(* Logix 5000 project; controller new_PLC_2 vendor 1 type 14 code 235 rev 37.11; software revision 37.00 *)

TASK MainTask (continuous, watchdog 500 ms) : MainProgram
TASK SafetyTask (periodic, rate 20 ms, priority 10, watchdog 20 ms, safety) : SafetyProgram

MODULES
   Local : vendor 1 type 14 code 235 (5069 0, rev 37.11)
      Tarjeta_Ethernet : vendor 1 type 12 code 200 (Ethernet 10.12.143.10, rev 10.7, Output RPI 10 ms)
           Point_IO_Gabinete_4:4:I   // Sensor Lane Change -
           Point_IO_Gabinete_2:4:O.3   // Stack Light Red
           Point_IO_Gabinete_2:4:O.1   // Stack Light Orange
           Point_IO_Gabinete_2:4:O.2   // Stack Light Green
           Point_IO_Gabinete_2:4:O   // Storage 2 Outputs Stack Lights
           Point_IO_Gabinete_4:8:O.2   // Cognex Light 2
           Point_IO_Gabinete_4:8:O.0   // Main Valve
           Point_IO_Gabinete_4:8:O.3   // Cognex Light 1
           Point_IO_Gabinete_4:8:O   // Main valve
           Point_IO_Gabinete_2:3:O.0   // Axis X -
           Point_IO_Gabinete_2:3:O.1   // Axis X +
           Point_IO_Gabinete_2:3:O.6   // Axis Y +
           Point_IO_Gabinete_2:3:O.2   // Gripper
           Point_IO_Gabinete_2:3:O.4   // Gripper Turn Conveyor
           Point_IO_Gabinete_2:3:O.3   // Gripper
           Point_IO_Gabinete_2:3:O.7   // Axis Y -
           Point_IO_Gabinete_2:3:O.5   // Gripper Turn Storage
           Point_IO_Gabinete_2:3:O   // Storage 2 Outputs
           Point_IO_Gabinete_4:7:O.6   // Lane Change 2
           Point_IO_Gabinete_4:7:O.7   // Lane Change 1
           Point_IO_Gabinete_4:7:O.0   // Pneumatic Cylinder 0
           Point_IO_Gabinete_4:7:O.1   // Pneumatic Cylinder 1
           Point_IO_Gabinete_4:7:O.2   // Pneumatic Cylinder 2
           Point_IO_Gabinete_4:7:O.3   // Pneumatic Cylinder 3
           Point_IO_Gabinete_4:7:O.4   // Pneumatic Cylinder D
           Point_IO_Gabinete_4:7:O.5   // Pneumatic Cylinder 4
           Point_IO_Gabinete_4:7:O   // Conveyor 2 Pneumatic Cylinders
           Point_IO_Gabinete_4:3:I.1   // Sensor Lane Change 1 +
           Point_IO_Gabinete_4:3:I.3   // Sensor Lane Change 2 -
           Point_IO_Gabinete_4:3:I.4   // Sensor Lane Change 1 -
           Point_IO_Gabinete_4:3:I.0   // Sensor Lane Change 2 +
           Point_IO_Gabinete_4:3:I   // Sensor Lane Change +
           Point_IO_Gabinete_2:1:I.6   // Sensor Gripper Turn Conveyor
           Point_IO_Gabinete_2:1:I.7   // Sensor Gripper Turn Storage
           Point_IO_Gabinete_2:1:I.1   // Sensor Axis X -
           Point_IO_Gabinete_2:1:I.3   // Sensor Axis X +
           Point_IO_Gabinete_2:1:I.0   // Sensor Gripper
           Point_IO_Gabinete_2:1:I.4   // Sensor Axis Y -
           Point_IO_Gabinete_2:1:I.2   // Sensor Gripper
           Point_IO_Gabinete_2:1:I.5   // Sensor Axis Y +
           Point_IO_Gabinete_2:1:I   // Storage 2 Inputs
           Point_IO_Gabinete_4:5:I.0   // Inductive Sensor 3
           Point_IO_Gabinete_4:5:I.1   // Inductive Sensor 5
           Point_IO_Gabinete_4:5:I.2   // Inductive Sensor 6
           Point_IO_Gabinete_4:5:I.3   // Inductive Sensor 4
           Point_IO_Gabinete_4:5:I.4   // Inductive Sensor 1
           Point_IO_Gabinete_4:5:I.5   // Inductive Sensor 2
           Point_IO_Gabinete_4:5:I   // Conveyor 2 Inductive Sensors
         @465399e0@:Partner : vendor 1 type 14 code 146 (ICP 2, rev 31.11)
         PLC_Safety : vendor 1 type 14 code 148 (ICP 1, rev 31.11, $3ebfc3d7$ RPI 20 ms)
      Variador_Conveyor_2 : PowerFlex 525-EENET (Ethernet 10.12.143.7, rev 5.1, Output RPI 20 ms)
      Camera_Conveyor_2 : vendor 678 type 100 code 260 (Ethernet 10.12.143.4, rev 12.1, Output RPI 60 ms)
      Point_IO_Gabinete_4 : 1734-AENTR (Ethernet 10.12.143.43, rev 5.12, Output RPI 20 ms)
         Modulo_Input_46 : 1734-IB8 (PointIO 6, rev 3.22)
         Modulo_Input_45 : 1734-IB8 (PointIO 5, rev 3.22)
         Modulo_Input_41 : 1734-IB8 (PointIO 1, rev 3.22)
         Modulo_Input_43 : 1734-IB8 (PointIO 3, rev 3.22)
         Modulo_Input_44 : 1734-IB8 (PointIO 4, rev 3.22)
         Modulo_Input_42 : 1734-IB8 (PointIO 2, rev 3.22)
         Modulo_Output_41 : 1734-OB8 (PointIO 7, rev 3.22)
         Modulo_Output_42 : 1734-OB8 (PointIO 8, rev 3.22)
         Modulo_Relay_42 : 1734-OW4 (PointIO 10, rev 3.22)
         Modulo_Relay_41 : 1734-OW4 (PointIO 9, rev 3.22)
      Point_IO_Gabinete_2 : 1734-AENTR (Ethernet 10.12.143.41, rev 5.12, Output RPI 20 ms)
         Modulo_Input_22 : 1734-IB8 (PointIO 2, rev 3.22)
         Modulo_Input_21 : 1734-IB8 (PointIO 1, rev 3.22)
         Modulo_Output_21 : 1734-OB8 (PointIO 3, rev 3.22)
         Modulo_Output_22 : 1734-OB8 (PointIO 4, rev 3.22)
         Modulo_Relay_2 : 1734-OW4 (PointIO 5, rev 3.22)
      PLC1 : vendor 1 type 14 code 235 (Ethernet 10.12.143.17, rev 37.11, $4f769f2f$ RPI 20 ms)
END_MODULES

VAR_GLOBAL   (* controller tags *)
   Contador_Prog : COUNTER;
   Data_from_PLC_1 : DINT[20] := ([1] := 130);
   Data_From_PLC_Safety : DINT[20] := ([0] := 1, [2] := 8388609);
        [0].0   // Safety_ok
   Data_to_PLC_1 : DINT[20]; {produced}
   Data_to_PLC_Safety : DINT[20]; {produced}
   E_0 : BOOL := 1;
   E_1 : BOOL;   // Estado1_PLC_2
   E_2 : BOOL;   // Estado2_PLC_2
   E_3 : BOOL;   // Estado3_PLC_2
   E_4 : BOOL;   // Estado4_PLC_2
   E_5 : BOOL;   // Estado5_PLC_2
   E_Stop_OK : BOOL := 1;
   Mult_prog : REAL := 12.5;
   Porcen_acum : REAL := 33.33;
   Safety_OK : BOOL := 1;
   Sgn_Rob : BOOL;
   Strt : BOOL;
   T0_1 : BOOL;
   T1_2 : BOOL;
   T2_3 : BOOL;
   T3_4 : BOOL;
   T4_5 : BOOL;
   T5_1 : BOOL;
   T5_6 : BOOL;
   T6_1 : BOOL;
   Timer1 : TIMER := (PRE := 2000);
   TimerCam : TIMER := (PRE := 5000);
   x : DINT;
END_VAR

PROGRAM MainProgram   (* main routine MainRoutine *)
VAR
   Ciclo_finalizado : BOOL;
   cleaning : BOOL;
   Contador_Piezas_salida : COUNTER := (PRE := 1);
   contador_triger : COUNTER := (CU := 1, DN := 1);
   paso0 : REAL;
   paso1 : REAL := 2.53;
   paso10 : REAL := 66.66;
   paso11 : REAL := 66.66;
   paso12 : REAL;
   paso13 : REAL := 73.32;
   paso14 : REAL := 79.92;
   paso15 : REAL := 86.58;
   paso16 : REAL := 93.64;
   paso17 : REAL := 100.0;
   paso2 : REAL := 5.06;
   paso3 : REAL := 33.33;
   paso3_1 : REAL := 10.12;
   paso4 : REAL := 12.65;
   paso5 : REAL := 15.18;
   paso6 : REAL := 17.71;
   paso6_1 : REAL := 20.24;
   paso7 : REAL := 22.77;
   paso8 : REAL := 25.3;
   paso9 : REAL := 30.36;
   Reset_auto : BOOL;
   Reset_m : BOOL;
   sTO : BOOL;
   Tiempo_Ciclo : TIMER := (PRE := 10000000);
   Tiempo_E1 : TIMER := (PRE := 10000000);
   Tiempo_E2 : TIMER := (PRE := 10000000);
   Tiempo_E3 : TIMER := (PRE := 10000000);
   Trig_1 : BOOL := 1;
   Trig_2 : BOOL := 1;
   Trig_3 : BOOL := 1;
   Triger1 : REAL;
   Triger2 : REAL;
   Triger3 : REAL;
END_VAR

ROUTINE Conveyor_plc2   (* ladder *)
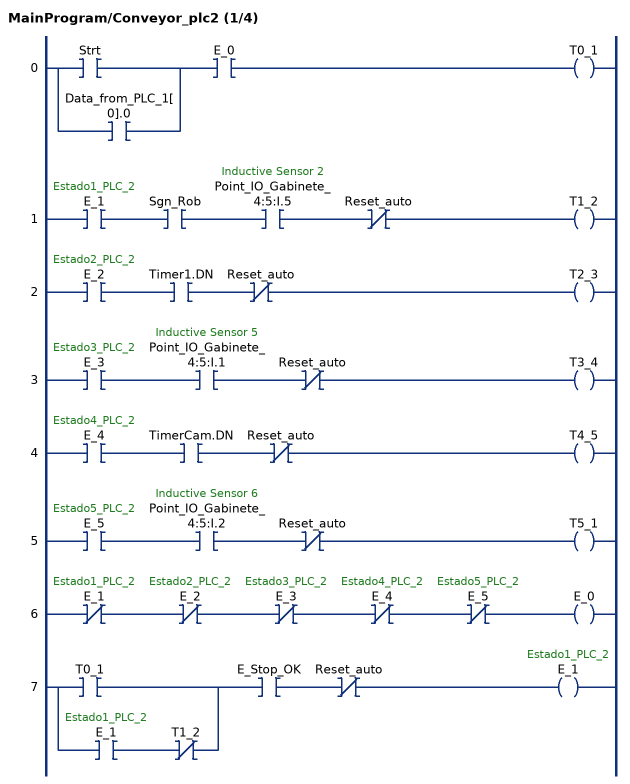
   0: [XIC(Strt) ,XIC(Data_from_PLC_1[0].0) ]XIC(E_0)OTE(T0_1);
   1: XIC(E_1)XIC(Sgn_Rob)XIC(Point_IO_Gabinete_4:5:I.5)XIO(Reset_auto)OTE(T1_2);
   2: XIC(E_2)XIC(Timer1.DN)XIO(Reset_auto)OTE(T2_3);
   3: XIC(E_3)XIC(Point_IO_Gabinete_4:5:I.1)XIO(Reset_auto)OTE(T3_4);
   4: XIC(E_4)XIC(TimerCam.DN)XIO(Reset_auto)OTE(T4_5);
   5: XIC(E_5)XIC(Point_IO_Gabinete_4:5:I.2)XIO(Reset_auto)OTE(T5_1);
   6: XIO(E_1)XIO(E_2)XIO(E_3)XIO(E_4)XIO(E_5)OTE(E_0);
   7: [XIC(T0_1) ,XIC(E_1) XIO(T1_2) ]XIC(E_Stop_OK)XIO(Reset_auto)OTE(E_1);
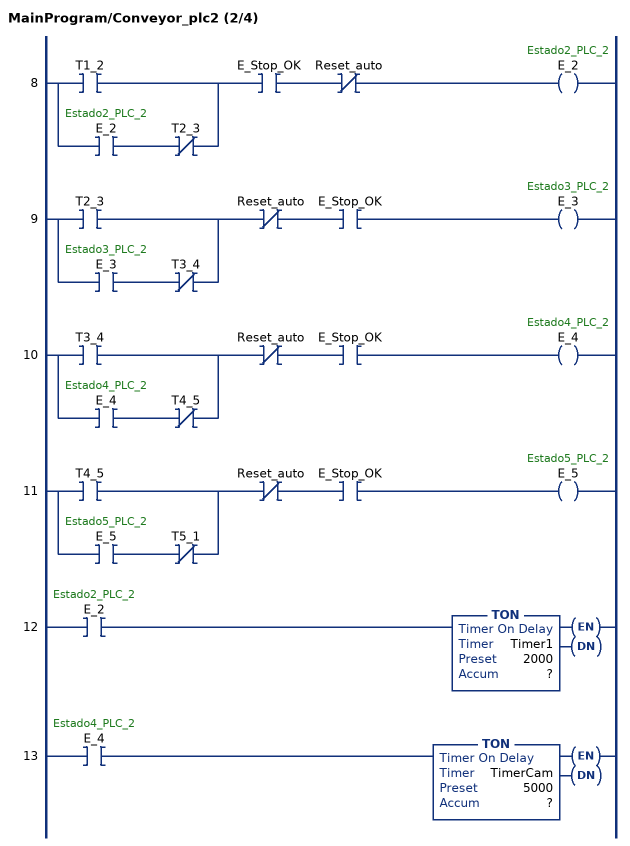
   8: [XIC(T1_2) ,XIC(E_2) XIO(T2_3) ]XIC(E_Stop_OK)XIO(Reset_auto)OTE(E_2);
   9: [XIC(T2_3) ,XIC(E_3) XIO(T3_4) ]XIO(Reset_auto)XIC(E_Stop_OK)OTE(E_3);
   10: [XIC(T3_4) ,XIC(E_4) XIO(T4_5) ]XIO(Reset_auto)XIC(E_Stop_OK)OTE(E_4);
   11: [XIC(T4_5) ,XIC(E_5) XIO(T5_1) ]XIO(Reset_auto)XIC(E_Stop_OK)OTE(E_5);
   12: XIC(E_2)TON(Timer1,?,?);
   13: XIC(E_4)TON(TimerCam,?,?);
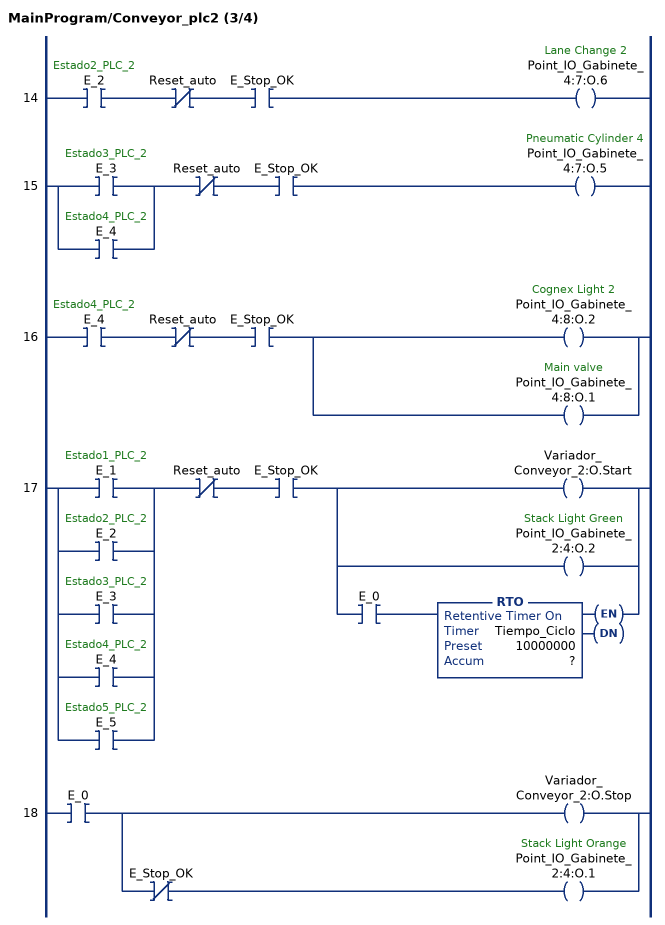
   14: XIC(E_2)XIO(Reset_auto)XIC(E_Stop_OK)OTE(Point_IO_Gabinete_4:7:O.6);
   15: [XIC(E_3) ,XIC(E_4) ]XIO(Reset_auto)XIC(E_Stop_OK)OTE(Point_IO_Gabinete_4:7:O.5);
   16: XIC(E_4)XIO(Reset_auto)XIC(E_Stop_OK)[OTE(Point_IO_Gabinete_4:8:O.2) ,OTE(Point_IO_Gabinete_4:8:O.1) ];
   17: [XIC(E_1) ,XIC(E_2) ,XIC(E_3) ,XIC(E_4) ,XIC(E_5) ]XIO(Reset_auto)XIC(E_Stop_OK)[OTE(Variador_Conveyor_2:O.Start) ,OTE(Point_IO_Gabinete_2:4:O.2) ,XIC(E_0) RTO(Tiempo_Ciclo,?,?) ];
   18: XIC(E_0)[OTE(Variador_Conveyor_2:O.Stop) ,XIO(E_Stop_OK) OTE(Point_IO_Gabinete_2:4:O.1) ];
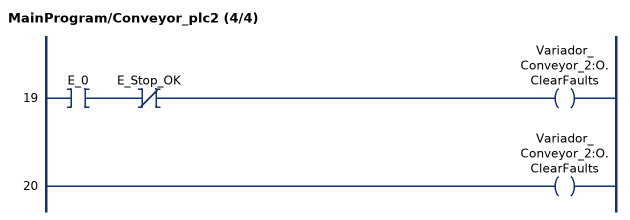
   19: XIC(E_0)XIO(E_Stop_OK)OTE(Variador_Conveyor_2:O.ClearFaults);
   20: OTE(Variador_Conveyor_2:O.ClearFaults);
END_ROUTINE

ROUTINE MainRoutine   (* ladder *)
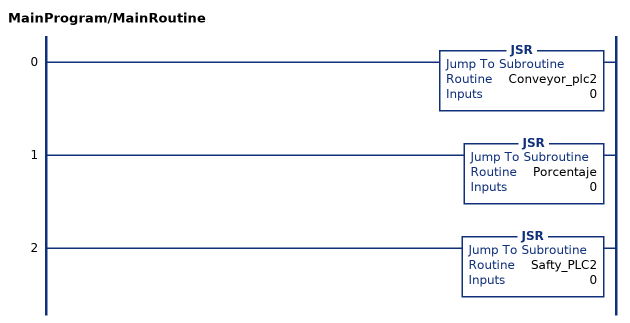
   0: JSR(Conveyor_plc2,0);
   1: JSR(Porcentaje,0);
   2: JSR(Safty_PLC2,0);
END_ROUTINE

ROUTINE Porcentaje   (* ladder *)
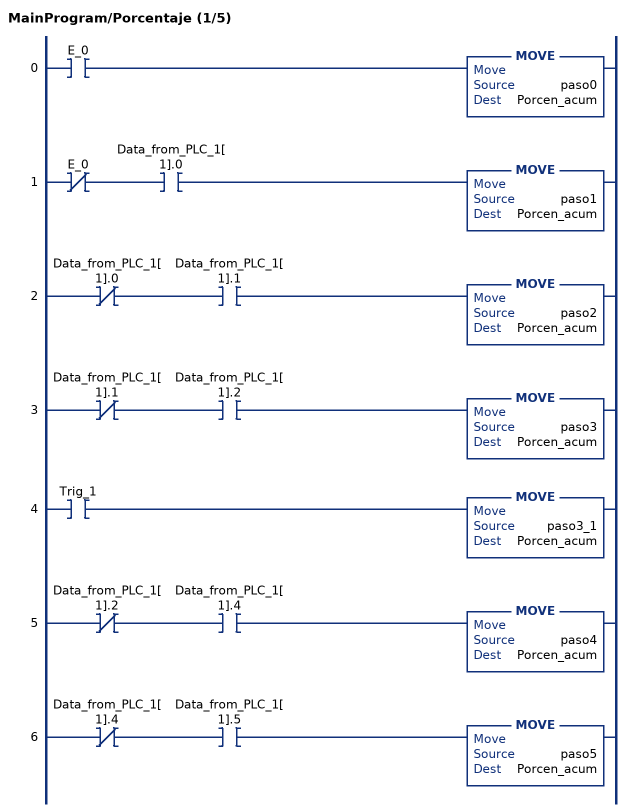
   0: XIC(E_0)MOVE(paso0,Porcen_acum);
   1: XIO(E_0)XIC(Data_from_PLC_1[1].0)MOVE(paso1,Porcen_acum);
   2: XIO(Data_from_PLC_1[1].0)XIC(Data_from_PLC_1[1].1)MOVE(paso2,Porcen_acum);
   3: XIO(Data_from_PLC_1[1].1)XIC(Data_from_PLC_1[1].2)MOVE(paso3,Porcen_acum);
   4: XIC(Trig_1)MOVE(paso3_1,Porcen_acum);
   5: XIO(Data_from_PLC_1[1].2)XIC(Data_from_PLC_1[1].4)MOVE(paso4,Porcen_acum);
   6: XIO(Data_from_PLC_1[1].4)XIC(Data_from_PLC_1[1].5)MOVE(paso5,Porcen_acum);
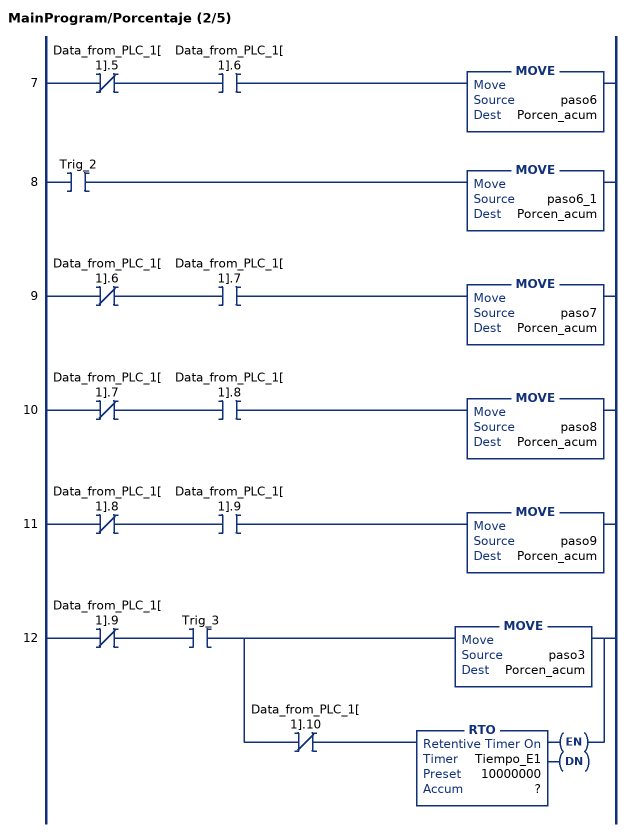
   7: XIO(Data_from_PLC_1[1].5)XIC(Data_from_PLC_1[1].6)MOVE(paso6,Porcen_acum);
   8: XIC(Trig_2)MOVE(paso6_1,Porcen_acum);
   9: XIO(Data_from_PLC_1[1].6)XIC(Data_from_PLC_1[1].7)MOVE(paso7,Porcen_acum);
   10: XIO(Data_from_PLC_1[1].7)XIC(Data_from_PLC_1[1].8)MOVE(paso8,Porcen_acum);
   11: XIO(Data_from_PLC_1[1].8)XIC(Data_from_PLC_1[1].9)MOVE(paso9,Porcen_acum);
   12: XIO(Data_from_PLC_1[1].9)XIC(Trig_3)[MOVE(paso3,Porcen_acum) ,XIO(Data_from_PLC_1[1].10) RTO(Tiempo_E1,?,?) ];
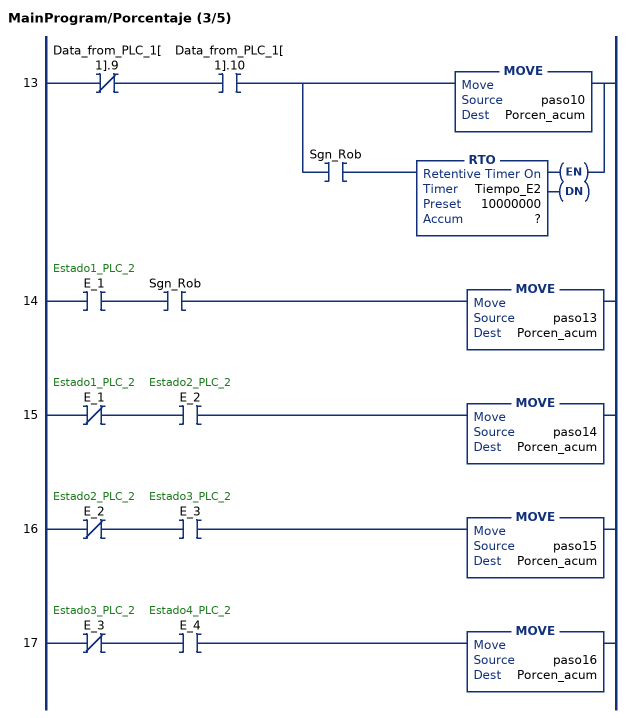
   13: XIO(Data_from_PLC_1[1].9)XIC(Data_from_PLC_1[1].10)[MOVE(paso10,Porcen_acum) ,XIC(Sgn_Rob) RTO(Tiempo_E2,?,?) ];
   14: XIC(E_1)XIC(Sgn_Rob)MOVE(paso13,Porcen_acum);
   15: XIO(E_1)XIC(E_2)MOVE(paso14,Porcen_acum);
   16: XIO(E_2)XIC(E_3)MOVE(paso15,Porcen_acum);
   17: XIO(E_3)XIC(E_4)MOVE(paso16,Porcen_acum);
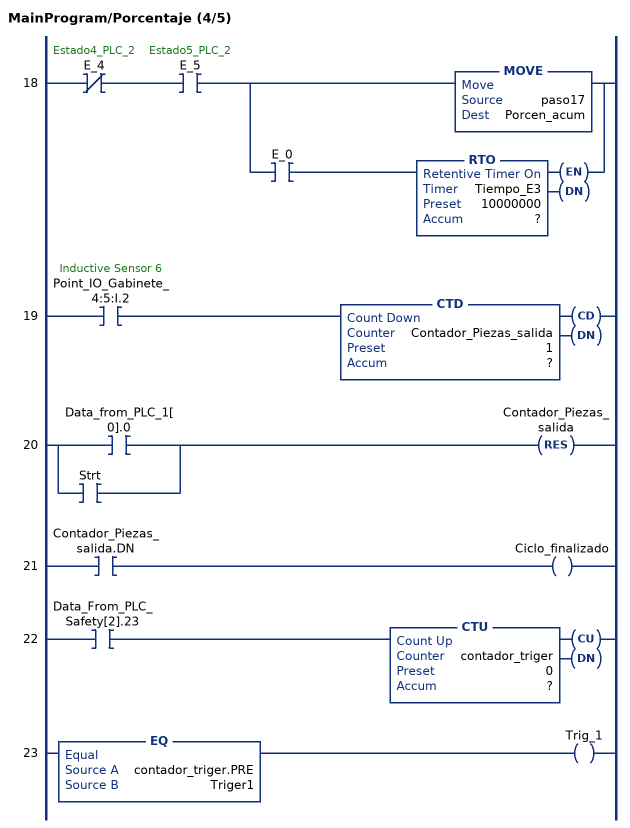
   18: XIO(E_4)XIC(E_5)[MOVE(paso17,Porcen_acum) ,XIC(E_0) RTO(Tiempo_E3,?,?) ];
   19: XIC(Point_IO_Gabinete_4:5:I.2)CTD(Contador_Piezas_salida,?,?);
   20: [XIC(Data_from_PLC_1[0].0) ,XIC(Strt) ]RES(Contador_Piezas_salida);
   21: XIC(Contador_Piezas_salida.DN)OTE(Ciclo_finalizado);
   22: XIC(Data_From_PLC_Safety[2].23)CTU(contador_triger,?,?);
   23: EQ(contador_triger.PRE,Triger1)OTE(Trig_1);
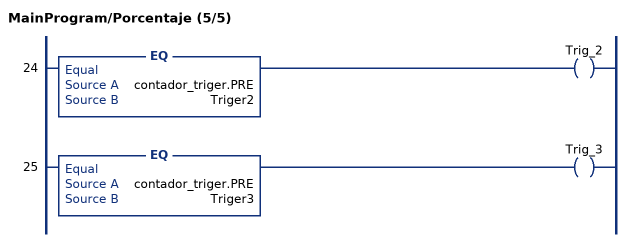
   24: EQ(contador_triger.PRE,Triger2)OTE(Trig_2);
   25: EQ(contador_triger.PRE,Triger3)OTE(Trig_3);
END_ROUTINE

ROUTINE Safty_PLC2   (* ladder *)
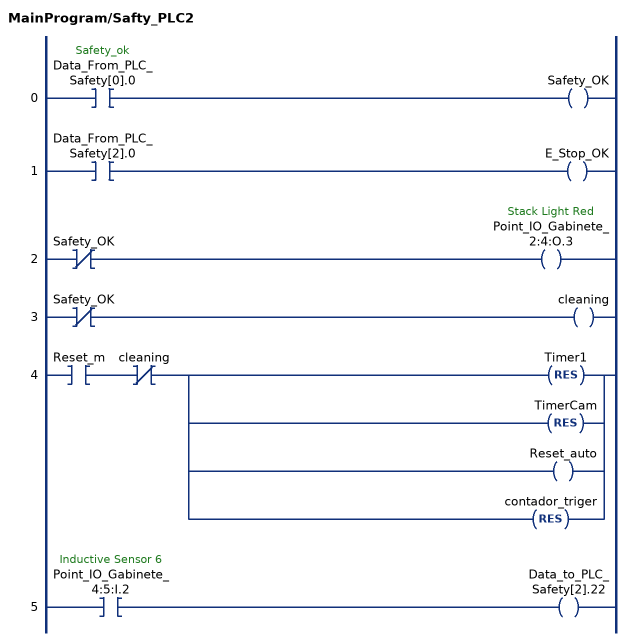
   0: XIC(Data_From_PLC_Safety[0].0)OTE(Safety_OK);
   1: XIC(Data_From_PLC_Safety[2].0)OTE(E_Stop_OK);
   2: XIO(Safety_OK)OTE(Point_IO_Gabinete_2:4:O.3);
   3: XIO(Safety_OK)OTE(cleaning);
   4: XIC(Reset_m)XIO(cleaning)[RES(Timer1) ,RES(TimerCam) ,OTE(Reset_auto) ,RES(contador_triger) ];
   5: XIC(Point_IO_Gabinete_4:5:I.2)OTE(Data_to_PLC_Safety[2].22);
END_ROUTINE
END_PROGRAM

PROGRAM SafetyProgram   (* main routine MainRoutine, safety *)

ROUTINE MainRoutine   (* ladder *)
END_ROUTINE
END_PROGRAM
